(* CoDeSys 2.3 export: LogLibBasic.EXP *)

(* Global variable list: basic/LogLibBasic *)
VAR_GLOBAL

    GlobalLogBufferHandle: LogBufferHandle;
    GlobalTick: UDINT;

END_VAR
